// TwinCAT 3 PLC project ConnectRobots
// Title: Mobile Manipulator Omron
// Company: Hochschule Luzern
// ProjectVersion: 0.0.0.1
// ProgramVersion: 3.1.4023.0
// libraries:
//   Tc2_ModbusSrv, * (Beckhoff Automation GmbH)
//   Tc2_Standard, * (Beckhoff Automation GmbH)
//   Tc2_System, * (Beckhoff Automation GmbH)
//   Tc2_TcpIp, * (Beckhoff Automation GmbH)
//   Tc2_Utilities, * (Beckhoff Automation GmbH)
//   Tc3_EventLogger, * (Beckhoff Automation GmbH)
//   Tc3_Module, * (Beckhoff Automation GmbH)
//   VisuDialogs, * (System)
//   Mobile Manipulator Omron,0.0.0.1,Hochschule Luzern
//   Tc2_OpcUa,3.3.2.0,Beckhoff Automation GmbH
// project tree:
//   / ClassDiagramTrial.TcCD (not stored), GlobalTextList.TcGTLO, PlcTask.TcTTO, Visualization Manager.TcVMO (not stored)
//   DUTs/ E_MoMa_2ndHierarchy_Implementation.TcDUT, E_MoMa_1stHierarchy_States.TcDUT
//   DUTs/LD_MobileRobot/ E_DataExchangeLD.TcDUT, ST_MobileRobotObjectLD.TcDUT
//   DUTs/TM_Manipulator/ E_CommandEventTM.TcDUT (not stored), ST_RobotArmObjectTM.TcDUT
//   GVLs/ GCL_TcpIp.TcGVL, GCL_ModbusTcp.TcGVL (not stored), GVL_CommandWindow.TcGVL, GVL_MobileManipulator.TcGVL
//   POUs/ FB_MobileManipulator9DoF.TcPOU, MAIN.TcPOU
//   POUs/LD_MobileRobot/ FB_HandleRobotLD.TcPOU (not stored), FB_SocketLD.TcPOU
//   POUs/TM_Manipulator/ FB_HandleGetTM.TcPOU (not stored), FB_HandleSetTM.TcPOU (not stored), FB_ModbusReadTM.TcPOU, FB_ModbusWriteTM.TcPOU (not stored)
//   VISUs/ CommandWindow.TcVIS
// real-time tasks:
//   TASK PlcTask: cycle T#10ms, priority 20, ADS port 350

CONFIGURATION ConnectRobots
    RESOURCE PLC ON TwinCAT3
        TASK PlcTask(INTERVAL := T#10ms, PRIORITY := 20);
        PROGRAM MAIN WITH PlcTask : MAIN;
    END_RESOURCE
END_CONFIGURATION

// ---- DUTs/E_MoMa_2ndHierarchy_Implementation.TcDUT
TYPE E_MoMa_2ndHierarchy_Implementation :
(
	Decision,
	MovingTM,
	MovingLD,
	VisionTask
)UDINT;
END_TYPE

// ---- DUTs/E_MoMa_1stHierarchy_States.TcDUT
TYPE E_MoMa_1stHierarchy_States :
(
	Init,
	IdleState,
	UserInteraction, 
	Prepare,
	Implementation,
	Clear,
	ServiceNeeded
)UDINT;
END_TYPE

// ---- DUTs/LD_MobileRobot/E_DataExchangeLD.TcDUT
TYPE E_DataExchangeLD :
(
	IDLE,
	ConnectServer,
	ExchangeData,
	Succeed,
	ERROR
)UDINT;
END_TYPE

// ---- DUTs/LD_MobileRobot/ST_MobileRobotObjectLD.TcDUT
{attribute 'OPC.UA.DA.StructuredType' := '1'}
TYPE ST_MobileRobotObjectLD :
STRUCT
	//'Status: Robot joystick driving StateOfCharge: 52.2 Location: 2867572 -89647 48 Temperature: 36$R$N'
	sStatus			: STRING;
	fBattery		: REAL;
	fPositionX  	: REAL;
	fPositionY 		: REAL;
	fRotationTheta 	: REAL; 
	nTemperature 	: INT;
	
	bBusyLD 	: BOOL; //TRUE: if moving, FALSE: if stable 
	bErrorLD	: BOOL; //TRUE: if error or cannot read the server, FALSE: reading status
END_STRUCT
END_TYPE

// ---- DUTs/TM_Manipulator/ST_RobotArmObjectTM.TcDUT
{attribute 'OPC.UA.DA.StructuredType' := '1'}
TYPE ST_RobotArmObjectTM :
STRUCT
	cmdID : E_CommandEventTM;

	fX : REAL; 
	fY : REAL; 
	fZ : REAL; 
	fRX : REAL; 
	fRY : REAL; 
	fRZ : REAL; 
	
	fTheta1 : REAL := 0;
	fTheta2 : REAL := 0;
	fTheta3 : REAL := 0;
	fTheta4 : REAL := 0;
	fTheta5 : REAL := 0;
	fTheta6 : REAL := 0;
	
	bBusyTM 	: BOOL; //TRUE: if project running, FALSE: not moving
	bErrorTM	: BOOL; //TRUE: error, FALSE: not
	
END_STRUCT
END_TYPE

// ---- GVLs/GCL_TcpIp.TcGVL
{attribute 'qualified_only'}
VAR_GLOBAL CONSTANT
	sSrvNetID		: T_AmsNetID	:= '';(* TwinCAT TCP/IP server network address *)
	sRemoteHost 	: T_IPv4Addr := '1.2.3.4';
	nRemotePort 	: UDINT:=7171;
END_VAR

// ---- GVLs/GVL_CommandWindow.TcGVL
{attribute 'qualified_only'}
VAR_GLOBAL
	
	(*--------------- TM5-700 Connection Parameters ---------------*)
	
	//methods
	bCmdMoveRelPTP : BOOL;
	bCmdMoveRelLinear : BOOL;
	bCmdSetJointsPTP : BOOL;

	
	fX_Ref : REAL;
	fY_Ref : REAL;
	fZ_Ref : REAL;
	fRX_Ref : REAL;
	fRY_Ref : REAL;
	fRZ_Ref : REAL;
	
	fTheta1_Ref : REAL;
	fTheta2_Ref : REAL;
	fTheta3_Ref : REAL;
	fTheta4_Ref : REAL;
	fTheta5_Ref : REAL;
	fTheta6_Ref : REAL;
	
	fX_Current : REAL;
	fY_Current : REAL;
	fZ_Current : REAL;
	fRX_Current : REAL;
	fRY_Current : REAL;
	fRZ_Current : REAL;
	
	fTheta1_Current : REAL;
	fTheta2_Current : REAL;
	fTheta3_Current : REAL;
	fTheta4_Current : REAL;
	fTheta5_Current : REAL;
	fTheta6_Current : REAL;
	
	commandID : E_CommandEventTM;
	
	
	
	(*--------------- LD-90 Connection Parameters ---------------*)
	bCmdWriteStringToLD90 : BOOL;
	
	sWriteCommand : STRING;
	
	//sReceivedCommands : ARRAY [0..20] OF STRING;
	sReceivedCommands : STRING(7680);
	
	
END_VAR

// ---- GVLs/GVL_MobileManipulator.TcGVL
{attribute 'qualified_only'}
VAR_GLOBAL
	
	(*--------------- Omron TM5 Manipulator Parameters  ---------------*)
	{attribute 'OPC.UA.DA' := '1'}
	bStartTM	: BOOL;
	{attribute 'OPC.UA.DA' := '1'}
	bStopTM		: BOOL;
	
	
	{attribute 'OPC.UA.DA' := '1'}
	stRobotArmObjectTM : ST_RobotArmObjectTM;
	
	

	
	
	
	(*--------------- Omron LD-90 Mobile Robot Parameters  ---------------*)
	{attribute 'OPC.UA.DA' := '1'}
	bStartLD 	: BOOL;
	{attribute 'OPC.UA.DA' := '1'}
	bStopLD		: BOOL;
	statusReceivedLD 	: STRING(7680):= '';
	statusWriteLD 		: T_MaxString; 
	
	{attribute 'OPC.UA.DA' := '1'}
	stMobileRobotObjectLD : ST_MobileRobotObjectLD;

 

END_VAR

// ---- POUs/MAIN.TcPOU
PROGRAM MAIN
VAR
	fbMobileManipulator9DoF : FB_MobileManipulator9DoF;
	
END_VAR

fbMobileManipulator9DoF();

END_PROGRAM

// ---- POUs/FB_MobileManipulator9DoF.TcPOU
FUNCTION_BLOCK FB_MobileManipulator9DoF
VAR_INPUT
END_VAR
VAR_OUTPUT
END_VAR
VAR
	
	//Initializing FuncBlock objects for LD-90 and TM5-700
	{attribute 'OPC.UA.DA':='1'}
	fbHandleRobotLD : FB_HandleRobotLD;
	{attribute 'OPC.UA.DA':='1'}
	fbHandleSetTM : FB_HandleSetTM;
	fbHandleGetTM : FB_HandleGetTM;
	
//	fbSetRobotTM 				: FB_SetRobotTM;	
//	fbReadRobotTM 			: FB_ReadRobotTM;
	
	
	// Variables to call LD class functions 
	{attribute 'OPC.UA.DA' := '1'}
    bLDgetRobotIP : BOOL;
	{attribute 'OPC.UA.DA' := '1'}
	sRobotIP : STRING;
	bLDgetTargetList : BOOL;
	bLDgetHomePos : BOOl;
	{attribute 'OPC.UA.DA' := '1'}
	bLDshutdown : BOOL;
	{attribute 'OPC.UA.DA' := '1'}
	stLDmobileRobotObject : ST_MobileRobotObjectLD;
	
	//Variables to call TM class functions
	{attribute 'OPC.UA.DA' := '1'}
	bTMbuttonPlayPause : BOOL;
	{attribute 'OPC.UA.DA' := '1'}
	bTMbuttonStop 	 : BOOL;
	{attribute 'OPC.UA.DA' := '1'}
	bTMmoveRelativePTP : BOOL;
	{attribute 'OPC.UA.DA' := '1'}
	bTMsetJointsPTP : BOOL;
	{attribute 'OPC.UA.DA' := '1'}
	stTMrobotArmObject : ST_RobotArmObjectTM;
	
	//State Machine 
	eState : E_MoMaStates;
END_VAR

(*--------------- Calling LD-90 handler & methods ---------------*)
//handler
fbHandleRobotLD();

//method: getRobotIP 
IF bLDgetRobotIP THEN
	fbHandleRobotLD.getRobotIP(bDone=>bLDgetRobotIP); 
	sRobotIP := fbHandleRobotLD.sGetRobotIP;
END_IF	
sRobotIP := fbHandleRobotLD.sGetRobotIP;

//method: shutdown
IF bLDshutdown THEN
	fbHandleRobotLD.shutdown(bDone=>bLDshutdown);
END_IF
(*--------------- END OF Calling LD-90 handler & methods ---------------*)



(*--------------- Calling TM5-700 handler & methods ---------------*)
//set handler
fbHandleSetTM();

//get handler
fbHandleGetTM();

//IF GVL_CommandWindow.bCmdMoveRelPTP THEN
//	fbSetRobotTM();
//END_IF

//method: buttonPlayPause
IF bTMbuttonPlayPause THEN
	bTMbuttonPlayPause := fbHandleSetTM.buttonPlayPause();
END_IF

//method: buttonStop
IF bTMbuttonStop THEN
	bTMbuttonStop := fbHandleSetTM.buttonStop();
END_IF

//method: moveRelativePTP
IF bTMmoveRelativePTP THEN
	bTMmoveRelativePTP := fbHandleSetTM.moveRelativePTP(stTMrobotArmObject.fX, stTMrobotArmObject.fY, stTMrobotArmObject.fZ, 
								  stTMrobotArmObject.fRX, stTMrobotArmObject.fRY, stTMrobotArmObject.fRZ);
END_IF

//method: setJointPTP
IF bTMsetJointsPTP THEN
	bTMsetJointsPTP := fbHandleSetTM.setJointsPTP(stTMrobotArmObject.fTheta1, stTMrobotArmObject.fTheta2, stTMrobotArmObject.fTheta3,
							   stTMrobotArmObject.fTheta4, stTMrobotArmObject.fTheta5, stTMrobotArmObject.fTheta6);
END_IF

(*--------------- END OF Calling TM5-700 handler & methods ---------------*)




(*--------------- TO DO: Task Separator for Robots to NOT Move Simultaniously ---------------*)
	
CASE eState OF
	Init:
		IF GVL_MobileManipulator.stMobileRobotObjectLD.bErrorLD OR  GVL_MobileManipulator.stRobotArmObjectTM.bErrorTM THEN
			eState := ServiceNeeded;	
		END_IF
	Prepare: 
		//prepare queue for the task 
		IF GVL_MobileManipulator.bStartTM THEN
			eState := Moving_TM;
		ELSIF GVL_MobileManipulator.bStartLD THEN
			eState := Moving_LD;
		END_IF
		
		//IF tasks are finished then
			eState := Succeeded;
		
	Moving_TM:
		GVL_MobileManipulator.bStopLD := TRUE; 
		//do what task requires
	
	Moving_LD:
		// move TM into embryo position 
		GVL_MobileManipulator.bStopTM := TRUE; 
		//do what task requires 
	Succeeded:
		eState := Init;
	
	Failed:
		// REprepare !!!
		eState := Prepare;

	ServiceNeeded:
		GVL_MobileManipulator.bStopTM := TRUE;
		GVL_MobileManipulator.bStopLD := TRUE;
END_CASE

END_FUNCTION_BLOCK

// ---- POUs/LD_MobileRobot/FB_SocketLD.TcPOU
//This function block creates a socket connection with the TCP/IP server of the mobile robot. It also handles the data exchange in terms of byte strings.
FUNCTION_BLOCK FB_SocketLD
VAR_INPUT
	//sWriteData : STRING :='';
	bStartWritingString : BOOL:=FALSE; //activated to send strings
END_VAR
VAR_OUTPUT
	//sReceivedCommands : STRING;
END_VAR
VAR
	eState: E_DataExchangeLD;
	kaanReceivedBytes : INT;
	
	//FB_SocketCloseAll 
	fbCloseAll		: FB_SocketCloseAll;
	bInitialize		: BOOL := TRUE;
	
	//FB_SocketConnect
	fbSocketConnect: FB_SocketConnect;
	bBusyConnect : BOOL;
	bErrorConnect : BOOL;
	hSocketConnect: Tc2_TcpIp.T_HSOCKET;
	nErrIdConnect: UDINT;
	bStart : BOOL:=TRUE;
	
	//FB_SocketReceive
	fbSocketReceive : FB_SocketReceive;
	arrDataReceive : ARRAY [0..7679] OF BYTE;
	bBusyReceive: BOOL;
	bErrorReceive: BOOL;
	nErrIdReceive: UDINT;
	nRecBytes: UDINT;
	
	//FB_SocketSend
	fbSocketSend : FB_SocketSend;
	arrDataSend : ARRAY [0..255] OF BYTE;
	bBusySend: BOOL;
	bErrorSend: BOOL;
	nErrIdSend: UDINT;
	
	//Connection Variables
	sSrvNetID		: T_AmsNetID	:= GCL_TcpIp.sSrvNetID;
	sRemoteHost 	: T_IPv4Addr := GCL_TcpIp.sRemoteHost;
	nRemotePort 	: UDINT:=GCL_TcpIp.nRemotePort;
	
	
	//Internal variables 
	i: INT;
	j : INT;
	k : INT;
	arrTmp : ARRAY [0..255] OF BYTE;
	sTmpMsg1 : STRING(255);
	sTmpMsg : T_MaxString;
	sTmpReceived : STRING(7680);
	
END_VAR



CASE eState OF
	IDLE:	
		(*--------------- On PLC close all previous connections ---------------*)
		fbCloseAll( sSrvNetID := sSrvNetID, bExecute:= bInitialize );
		IF fbCloseAll.bBusy OR fbCloseAll.bError THEN
			RETURN; // i don't like return
		END_IF
		bInitialize := FALSE;
		eState := ConnectServer;
		
		
	
	ConnectServer:
	
		(*--------------- Connect to the server  ---------------*)
		fbSocketConnect(
			sSrvNetID:=sSrvNetID, sRemoteHost:=sRemoteHost, nRemotePort:= nRemotePort, bExecute := TRUE, tTimeout := T#1S,
			bBusy => bBusyConnect, bError => bErrorConnect, nErrId => nErrIdConnect, hSocket => hSocketConnect);
		IF NOT fbSocketConnect.bBusy AND NOT fbSocketConnect.bError THEN
			fbSocketConnect.bExecute := FALSE;
			eState := ExchangeData;
		ELSIF fbSocketConnect.bError THEN
			eState := ERROR;
		END_IF
		IF fbSocketConnect.bBusy THEN
			eState := IDLE;
		END_IF
				
	ExchangeData:
	
		(*--------------- Get LD-90 String Commands ---------------*)
		
		
		//Receive Data
		fbSocketReceive(
			sSrvNetID :=sSrvNetID, hSocket := hSocketConnect, cbLen := SIZEOF(arrDataReceive), pDest := ADR(arrDataReceive), bExecute := TRUE, tTimeout := T#1S,
			bBusy => bBusyReceive, bError => bErrorReceive, nErrId => nErrIdReceive, nRecBytes => nRecBytes);
			
		
		IF NOT fbSocketReceive.bBusy THEN
			fbSocketReceive(bExecute := FALSE);
		END_IF
			
		IF fbSocketReceive.bError THEN
			eState := ERROR;
			kaanReceivedBytes := 3;
		END_IF
		IF fbSocketReceive.nRecBytes > 2 THEN
			//kaanReceivedBytes := UDINT_TO_INT(fbSocketReceive.nRecBytes);
			sTmpReceived := '';
			FOR i:=0 TO 28 DO
				FOR j:= 0 TO 255 DO
					arrTmp[j] := arrDataReceive[i*256 + j];
				END_FOR
				sTmpMsg :=  BYTEARR_TO_MAXSTRING(arrTmp);
				CONCAT2(ADR(sTmpReceived), ADR(sTmpMsg),ADR(sTmpReceived), SIZEOF(sTmpReceived)-1);
			END_FOR
			GVL_MobileManipulator.statusReceivedLD := sTmpReceived;
			
			//update the command window for all except status 
			IF NOT (LEFT(GVL_MobileManipulator.statusReceivedLD,6) = 'Status') THEN
				GVL_CommandWindow.sReceivedCommands := GVL_MobileManipulator.statusReceivedLD;
			END_IF
			
				
		END_IF
					
		
		(*--------------- Set LD-90 String Command ---------------*)
		IF bStartWritingString THEN
			bStartWritingString := FALSE;
			MEMSET(ADR(arrDataReceive), 0 , SIZEOF(arrDataReceive)-1);
			MEMSET(ADR(arrDataSend),16#00,SIZEOF(arrDataSend));
			MEMSET(ADR(arrTmp),16#00,SIZEOF(arrTmp));
			arrDataSend[SIZEOF(arrDataSend) - 1] := 16#00;
			sTmpMsg1 := CONCAT(GVL_MobileManipulator.statusWriteLD, '$0A');
			arrTmp := MAXSTRING_TO_BYTEARR(sTmpMsg1);
			FOR k:=0 TO UINT_TO_INT(SIZEOF(arrDataSend))-1 DO
				IF k < UINT_TO_INT(SIZEOF(arrTmp)) THEN
					arrDataSend[k] := arrTmp[k];
				ELSE
					arrDataSend[k] := 16#00;
				END_IF
			END_FOR
			fbSocketSend.bExecute := TRUE;	
		END_IF
		
		fbSocketSend(
				sSrvNetID :=sSrvNetID, hSocket := hSocketConnect, cbLen := INT_TO_UDINT(LEN(sTmpMsg1)), pSrc := ADR(arrDataSend), tTimeout := T#1S,
				bBusy => bBusySend, bError => bErrorSend, nErrId => nErrIdSend);
		
			
				
		IF NOT fbSocketSend.bBusy THEN
			fbSocketSend(bExecute:=FALSE);
		END_IF
		
		IF fbSocketSend.bError THEN
			eState := ERROR;
			kaanReceivedBytes := 4;
		END_IF
			
	Succeed:
		kaanReceivedBytes:= 5;//here we could do sth
	ERROR:
		i := 2;//NOT GOOD, replace later
END_CASE

END_FUNCTION_BLOCK

// ---- POUs/TM_Manipulator/FB_ModbusReadTM.TcPOU
//This function block calls the Modbus Read functions with given addresses. It returns the values read in that memory locations. 
FUNCTION_BLOCK FB_ModbusReadTM
VAR_INPUT
	nMBAddr2	: WORD := 16#1C21; //Modbus address to read inputs (FC: 2)
	nMBAddr4	: WORD := 16#1B59; //Modbus address to read input registers (FC: 4)
END_VAR
VAR_OUTPUT
	fX : REAL; // X (Cartesian coordinate w.r.t. current Base without tool)
	fY : REAL; // Y (Cartesian coordinate w.r.t. current Base without tool)
	fZ : REAL; // Z (Cartesian coordinate w.r.t. current Base without tool)
	fRX : REAL; // Rx (Cartesian coordinate w.r.t. current Base without tool)
	fRY : REAL; // Ry (Cartesian coordinate w.r.t. current Base without tool)
	fRZ : REAL; // Rz (Cartesian coordinate w.r.t. current Base without tool)
	
	fTheta1 : REAL; // Joint 1
	fTheta2 : REAL; // Joint 2
	fTheta3 : REAL; // Joint 3
	fTheta4 : REAL; // Joint 4
	fTheta5 : REAL; // Joint 5
	fTheta6 : REAL; // Joint 6
	
	bError : BOOL; // TRUE: Error, FALSE: Not
	bProjectRunning : BOOL; // TRUE: Project Running, FALSE: Not
END_VAR
VAR
	arrTemp : ARRAY [0..1] OF WORD;
	
	//Modbus Variables - FC:2 Read Inputs
	fbRead2				: FB_MBReadInputs;
	bStart2				: BOOL;
	arrReadInputs 		: ARRAY [0..1] OF BYTE;
	nquantity2			: WORD := INT_TO_WORD(SIZEOF(arrReadInputs)/2);
	bBusy2				: BOOL;
	bError2				: BOOL;
	nErrId2				: UDINT;
	cbRead2				: UDINT;
	
	//Modbus Variables - FC:4 Read Input Registers
	fbRead4				: FB_MBReadInputRegs;
	bStart4				: BOOL;
	arrReadRegisters 	: ARRAY [0..23] OF WORD;
	nQuantity4			: WORD := INT_TO_WORD(SIZEOF(arrReadRegisters)/2);
	bBusy4				: BOOL;
	bError4				: BOOL;
	nErrId4				: UDINT;
	cbRead4				: UDINT;
	
	//General TM5 Modbus variables
	sIPAddr				: STRING(15) := GCL_ModbusTcp.cIPAddr;
	nTCPPort			: UINT := GCL_ModbusTcp.cTCPPort;
	nUnitID				: BYTE := GCL_ModbusTcp.cUnitID;
END_VAR


(*---------------Modbus function 2 - ReadInputs---------------*)
IF NOT bstart2 THEN	
	bStart2 := TRUE;
	fbRead2.bExecute := TRUE;
ELSE
	IF NOT fbRead2.bBUSY THEN
		bStart2 := FALSE;
	END_IF
	fbRead2.bExecute := FALSE;
END_IF
fbRead2(sIPAddr:= sIPAddr, nTCPPort:= nTCPPort, nUnitID:= nUnitID, nQuantity:= nQuantity2, nMBAddr:= nMBAddr2, cbLength:= SIZEOF(arrReadInputs) , 
	pDestAddr:= ADR(arrReadInputs), bExecute:= bStart2 , tTimeout:= T#1S, bBusy=>bBusy2, bError=> bError4, nErrId=> nErrId2, cbRead=> cbRead4 );
(*---------------END OF Modbus function 2 - ReadInputs---------------*)


(*---------------Modbus function 4 - ReadInputRegs---------------*)
IF NOT bstart4 THEN	
	bStart4 := TRUE;
	fbRead4.bExecute := TRUE;
ELSE
	IF NOT fbRead4.bBUSY THEN
		bStart4 := FALSE;
	END_IF
	fbRead4.bExecute := FALSE;
END_IF
fbRead4(sIPAddr:= sIPAddr, nTCPPort:= nTCPPort, nUnitID:= nUnitID, nQuantity:= nQuantity4, nMBAddr:= nMBAddr4, cbLength:= SIZEOF(arrReadRegisters) , 
	pDestAddr:= ADR(arrReadRegisters), bExecute:= bStart4 , tTimeout:= T#1S, bBusy=>bBusy4, bError=> bError4, nErrId=> nErrId4, cbRead=> cbRead4 );
(*---------------END OF Modbus function 4 - ReadInputRegs---------------*)
	

(*---------------Extract Read Inputs (Error, Project Running) ---------------*)
//bError := arrReadRegisters[0];
//bProjectRunning := arrReadRegisters[1];
(*---------------END OF Extract Read Inputs---------------*)


(*---------------Extract Read Input Registers (Cartesian and Joint Space Positions) ---------------*)
arrTemp[1] := arrReadRegisters[0];
arrTemp[0] := arrReadRegisters[1];
MEMCPY(ADR(fX), ADR(arrTemp), 4);  //xPos
arrTemp[1] := arrReadRegisters[2];
arrTemp[0] := arrReadRegisters[3];
MEMCPY(ADR(fY), ADR(arrTemp), 4);  //yPos
arrTemp[1] := arrReadRegisters[4];
arrTemp[0] := arrReadRegisters[5];
MEMCPY(ADR(fZ), ADR(arrTemp), 4);  //zPos
arrTemp[1] := arrReadRegisters[6];
arrTemp[0] := arrReadRegisters[7];
MEMCPY(ADR(fRX), ADR(arrTemp), 4);  //xRot
arrTemp[1] := arrReadRegisters[8];
arrTemp[0] := arrReadRegisters[9];
MEMCPY(ADR(fRY), ADR(arrTemp), 4);  //yRot
arrTemp[1] := arrReadRegisters[10];
arrTemp[0] := arrReadRegisters[11];
MEMCPY(ADR(fRZ), ADR(arrTemp), 4);  //zRot
arrTemp[1] := arrReadRegisters[12];
arrTemp[0] := arrReadRegisters[13];
MEMCPY(ADR(fTheta1), ADR(arrTemp), 4);  // joint 1
arrTemp[1] := arrReadRegisters[14];
arrTemp[0] := arrReadRegisters[15];
MEMCPY(ADR(fTheta2), ADR(arrTemp), 4);  // joint 2
arrTemp[1] := arrReadRegisters[16];
arrTemp[0] := arrReadRegisters[17];
MEMCPY(ADR(fTheta3), ADR(arrTemp), 4);  // joint 3
arrTemp[1] := arrReadRegisters[18];
arrTemp[0] := arrReadRegisters[19];
MEMCPY(ADR(fTheta4), ADR(arrTemp), 4);  // joint 4
arrTemp[1] := arrReadRegisters[20];
arrTemp[0] := arrReadRegisters[21];
MEMCPY(ADR(fTheta5), ADR(arrTemp), 4);  // joint 5
arrTemp[1] := arrReadRegisters[22];
arrTemp[0] := arrReadRegisters[23];
MEMCPY(ADR(fTheta6), ADR(arrTemp), 4);  // joint 6
(*---------------END OF Extract Read Input Registers---------------*)

END_FUNCTION_BLOCK

// ---- GlobalTextList.TcGTLO
TEXTLIST GlobalTextList
  902 = '%.0f'
  769 = '%.1f'
  270 = '%.2f'
  707 = '%1.f'
  880 = '%f'
  475 = '%i'
  381 = '%n'
  339 = '%s'
  527 = '@:'
  465 = 'Actual Values '
  699 = 'Battery:'
  627 = 'deg'
  516 = 'Joint 1:'
  80 = 'Joint 2:'
  60 = 'Joint 3:'
  571 = 'Joint 4:'
  778 = 'Joint 5:'
  477 = 'Joint 6:'
  117 = 'LD-90 Mobile Robot'
  967 = 'Load Home Position'
  726 = 'mm'
  610 = 'Move Robot Position'
  831 = 'MoveAbsolutePTP'
  116 = 'MoveRelativeLinear'
  78 = 'MoveRelativePTP'
  313 = 'only working one'
  871 = 'Position'
  266 = 'Position:'
  890 = 'R:'
  806 = 'Received Commands:'
  885 = 'Reset'
  952 = 'Reset '
  215 = 'RX:'
  585 = 'RY:'
  137 = 'RZ:'
  575 = 'Send'
  535 = 'Set Robot Joints'
  439 = 'SetJointsLinear'
  144 = 'SetJointsPTP'
  994 = 'Status:'
  316 = 'Temperature:'
  566 = 'TM5-700 Robot Arm'
  259 = 'Write Commands:'
  312 = 'X:'
  583 = 'Y:'
  639 = 'Z:'
END_TEXTLIST

// ---- VISUs/CommandWindow.TcVIS
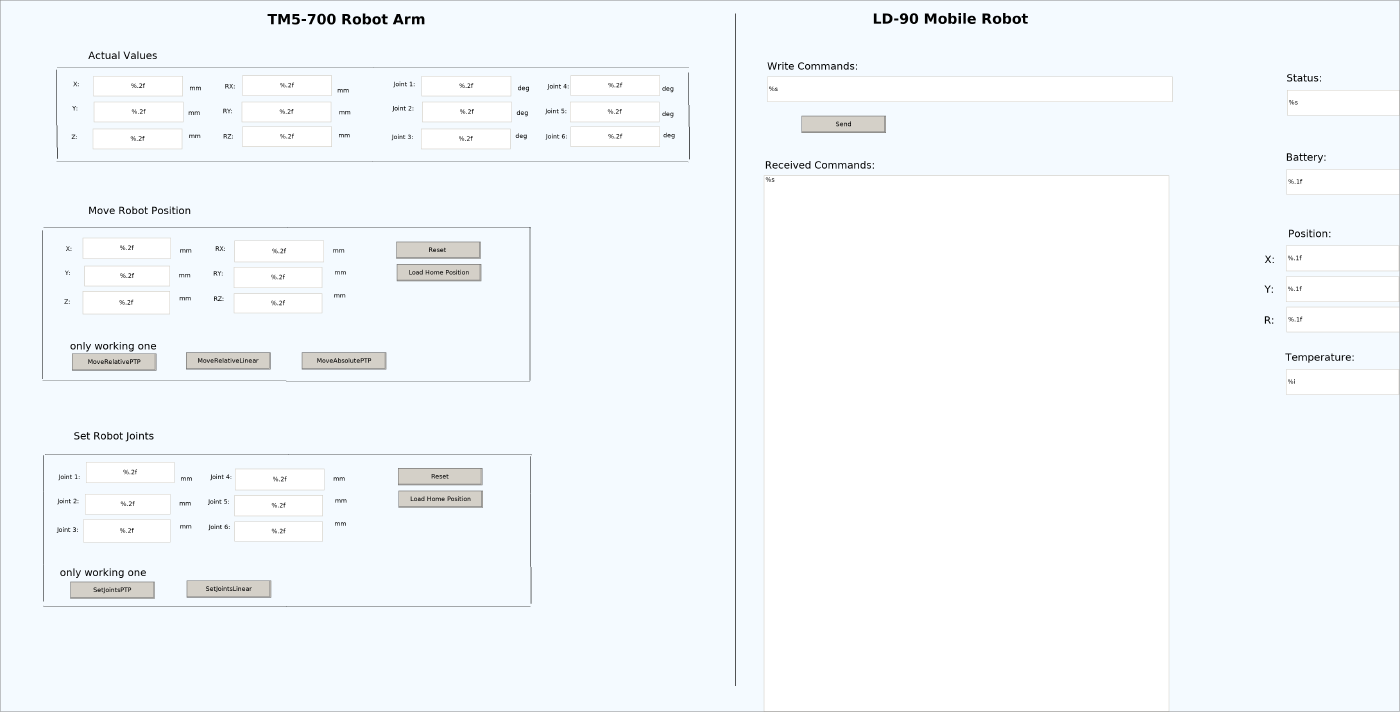
VISUALIZATION CommandWindow  // 2491x1267
    Textfield (147,423 157x37), "%.2f", text variable: GVL_CommandWindow.fX_Ref
        OnMouseClick: write the text variable via Default
    Textfield (150,473 152x36), "%.2f", text variable: GVL_CommandWindow.fY_Ref
        OnMouseClick: write the text variable via Default
    Textfield (147,518 155x41), "%.2f", text variable: GVL_CommandWindow.fZ_Ref
        OnMouseClick: write the text variable via Default
    Textfield (417,428 159x38), "%.2f", text variable: GVL_CommandWindow.fRX_Ref
        OnMouseClick: write the text variable via Default
    Textfield (416,475 157x37), "%.2f", text variable: GVL_CommandWindow.fRY_Ref
        OnMouseClick: write the text variable via Default
    Textfield (416,522 157x35), "%.2f", text variable: GVL_CommandWindow.fRZ_Ref
        OnMouseClick: write the text variable via Default
    Textfield (166,135 159x36), "%.2f", text variable: GVL_MobileManipulator.stRobotArmObjectTM.fX
    Textfield (167,181 159x36), "%.2f", text variable: GVL_MobileManipulator.stRobotArmObjectTM.fY
    Textfield (165,229 159x36), "%.2f", text variable: GVL_MobileManipulator.stRobotArmObjectTM.fZ
    Textfield (431,134 159x36), "%.2f", text variable: GVL_CommandWindow.fRX_Current
    Textfield (430,181 159x36), "%.2f", text variable: GVL_MobileManipulator.stRobotArmObjectTM.fRY
    Textfield (431,225 159x36), "%.2f", text variable: GVL_MobileManipulator.stRobotArmObjectTM.fRZ
    Label (109,133 53x34), "X:"
    Label (107,176 53x34), "Y:"
    Label (106,227 53x34), "Z:"
    Label (383,137 53x34), "RX:"
    Label (379,181 53x34), "RY:"
    Label (380,226 53x34), "RZ:"
    Label (334,142 40x30), "mm"
    Label (332,186 40x30), "mm"
    Label (333,227 40x30), "mm"
    Label (597,146 40x30), "mm"
    Label (600,185 40x30), "mm"
    Label (599,226 40x30), "mm"
    Label (85,82 273x34), "Actual Values"
    Label (83,358 331x34), "Move Robot Position"
    Textfield (750,135 159x36), "%.2f", text variable: GVL_MobileManipulator.stRobotArmObjectTM.fTheta1
    Textfield (751,181 159x36), "%.2f", text variable: GVL_MobileManipulator.stRobotArmObjectTM.fTheta2
    Textfield (749,229 159x36), "%.2f", text variable: GVL_MobileManipulator.stRobotArmObjectTM.fTheta3
    Textfield (1015,134 159x36), "%.2f", text variable: GVL_MobileManipulator.stRobotArmObjectTM.fTheta4
    Textfield (1014,181 159x36), "%.2f", text variable: GVL_MobileManipulator.stRobotArmObjectTM.fTheta5
    Textfield (1015,225 159x36), "%.2f", text variable: GVL_MobileManipulator.stRobotArmObjectTM.fTheta6
    Label (693,133 53x34), "Joint 1:"
    Label (691,176 53x34), "Joint 2:"
    Label (690,227 53x34), "Joint 3:"
    Label (967,137 53x34), "Joint 4:"
    Label (963,181 53x34), "Joint 5:"
    Label (964,226 53x34), "Joint 6:"
    Label (918,142 40x30), "deg"
    Label (916,186 40x30), "deg"
    Label (914,227 40x30), "deg"
    Label (1175,143 40x30), "deg"
    Label (1175,188 40x30), "deg"
    Label (1177,226 40x30), "deg"
    Label (96,426 53x34), "X:"
    Label (94,469 53x34), "Y:"
    Label (93,520 53x34), "Z:"
    Label (366,426 53x34), "RX:"
    Label (362,470 53x34), "RY:"
    Label (363,515 53x34), "RZ:"
    Label (317,431 40x30), "mm"
    Label (315,475 40x30), "mm"
    Label (316,516 40x30), "mm"
    Label (589,431 40x30), "mm"
    Label (592,470 40x30), "mm"
    Label (591,511 40x30), "mm"
    Button (128,629 150x30), "MoveRelativePTP"
        tap GVL_CommandWindow.bCmdMoveRelPTP
        OnMouseClick: execute { GVL_CommandWindow.commandID := MoveCartesianPTP; }
    Button (331,627 150x30), "MoveRelativeLinear"
        tap GVL_CommandWindow.bCmdMoveRelLinear
        OnMouseClick: execute { GVL_CommandWindow.commandID := MoveCartesianLine; }
    Button (537,627 150x30), "MoveAbsolutePTP"
    Button (706,470 150x30), "Load Home Position"
        OnMouseClick: execute {
            GVL_CommandWindow.fX_Ref := 100;
            GVL_CommandWindow.fY_Ref := 100;
            GVL_CommandWindow.fZ_Ref := 100;
            GVL_CommandWindow.fRX_Ref := 0;
            GVL_CommandWindow.fRY_Ref := 0;
            GVL_CommandWindow.fRZ_Ref := 90;
        }
    Textfield (153,822 157x37), "%.2f", text variable: GVL_CommandWindow.fTheta1_Ref
        OnMouseClick: write the text variable via Default
    Textfield (151,879 152x36), "%.2f", text variable: GVL_CommandWindow.fTheta2_Ref
        OnMouseClick: write the text variable via Default
    Textfield (148,924 155x41), "%.2f", text variable: GVL_CommandWindow.fTheta3_Ref
        OnMouseClick: write the text variable via Default
    Textfield (418,834 159x38), "%.2f", text variable: GVL_CommandWindow.fTheta4_Ref
        OnMouseClick: write the text variable via Default
    Textfield (417,881 157x37), "%.2f", text variable: GVL_CommandWindow.fTheta5_Ref
        OnMouseClick: write the text variable via Default
    Textfield (417,928 157x35), "%.2f", text variable: GVL_CommandWindow.fRZ_Ref
        OnMouseClick: write the text variable via Default
    Label (97,832 53x34), "Joint 1:"
    Label (95,875 53x34), "Joint 2:"
    Label (94,926 53x34), "Joint 3:"
    Label (367,832 53x34), "Joint 4:"
    Label (363,876 53x34), "Joint 5:"
    Label (364,921 53x34), "Joint 6:"
    Label (318,837 40x30), "mm"
    Label (316,881 40x30), "mm"
    Label (317,922 40x30), "mm"
    Label (590,837 40x30), "mm"
    Label (593,876 40x30), "mm"
    Label (592,917 40x30), "mm"
    Button (125,1035 150x30), "SetJointsPTP"
        tap GVL_CommandWindow.bCmdSetJointsPTP
        OnMouseClick: execute { GVL_CommandWindow.commandID := SetJointPositions; }
    Button (332,1033 150x30), "SetJointsLinear"
    Button (708,833 150x30), "Reset"
        OnMouseClick: execute {
            GVL_CommandWindow.fTheta1_Ref := 0;
            GVL_CommandWindow.fTheta2_Ref := 0;
            GVL_CommandWindow.fTheta3_Ref := 0;
            GVL_CommandWindow.fTheta4_Ref := 0;
            GVL_CommandWindow.fTheta5_Ref := 0;
            GVL_CommandWindow.fTheta6_Ref := 0;
        }
    Label (37,759 331x34), "Set Robot Joints"
    Button (705,430 150x30), "Reset"
        OnMouseClick: execute {
            GVL_CommandWindow.fX_Ref := 0;
            GVL_CommandWindow.fY_Ref := 0;
            GVL_CommandWindow.fZ_Ref := 0;
            GVL_CommandWindow.fRX_Ref := 0;
            GVL_CommandWindow.fRY_Ref := 0;
            GVL_CommandWindow.fRZ_Ref := 0;
        }
    Button (709,873 150x30), "Load Home Position"
        OnMouseClick: execute {
            GVL_CommandWindow.fTheta1_Ref := 0;
            GVL_CommandWindow.fTheta2_Ref := 90;
            GVL_CommandWindow.fTheta3_Ref := 0;
            GVL_CommandWindow.fTheta4_Ref := 0;
            GVL_CommandWindow.fTheta5_Ref := 0;
            GVL_CommandWindow.fTheta6_Ref := 0;
        }
    Label (36,599 331x34), "only working one"
    Label (18,1002 331x34), "only working one"
    Textfield (1359,312 721x955), "%s", text variable: GVL_CommandWindow.sReceivedCommands
    Label (1358,279 252x30), "Received Commands:"
    Textfield (1365,136 721x45), "%s", text variable: GVL_CommandWindow.sWriteCommand
        OnMouseClick: write the text variable via Default
    Label (1362,103 219x30), "Write Commands:"
    Button (1426,206 150x30), "Send"
        tap GVL_CommandWindow.bCmdWriteStringToLD90
    Line (101,287) (1224,288)
    Line (1309,1220) (1309,24)
    Line (1227,283) (1225,129)
    Line (102,119) (1225,120)
    Line (102,282) (100,124)
    Label (480,17 273x34), "TM5-700 Robot Arm"
    Label (1555,16 273x34), "LD-90 Mobile Robot"
    Line (76,674) (76,410)
    Line (76,677) (942,678)
    Line (78,404) (944,405)
    Line (80,808) (946,809)
    Line (77,1078) (943,1079)
    Line (943,677) (943,404)
    Line (78,1070) (77,810)
    Line (945,1074) (944,812)
    Textfield (2290,160 201x45), "%s", text variable: GVL_MobileManipulator.stMobileRobotObjectLD.sStatus
        OnMouseClick: write the text variable via Default
    Label (2286,124 117x30), "Status:"
    Textfield (2289,301 201x45), "%.1f", text variable: GVL_MobileManipulator.stMobileRobotObjectLD.fBattery
        OnMouseClick: write the text variable via Default
    Label (2285,265 117x30), "Battery:"
    Textfield (2288,437 201x45), "%.1f", text variable: GVL_MobileManipulator.stMobileRobotObjectLD.fPositionX
        OnMouseClick: write the text variable via Default
    Label (2289,401 117x30), "Position:"
    Textfield (2288,492 201x45), "%.1f", text variable: GVL_MobileManipulator.stMobileRobotObjectLD.fPositionY
        OnMouseClick: write the text variable via Default
    Textfield (2289,546 201x45), "%.1f", text variable: GVL_MobileManipulator.stMobileRobotObjectLD.fRotationTheta
        OnMouseClick: write the text variable via Default
    Textfield (2288,657 201x45), "%i", text variable: GVL_MobileManipulator.stMobileRobotObjectLD.nTemperature
        OnMouseClick: write the text variable via Default
    Label (2284,621 117x30), "Temperature:"
    Label (2247,447 28x30), "X:"
    Label (2247,500 28x30), "Y:"
    Label (2246,555 28x30), "R:"
END_VISUALIZATION
